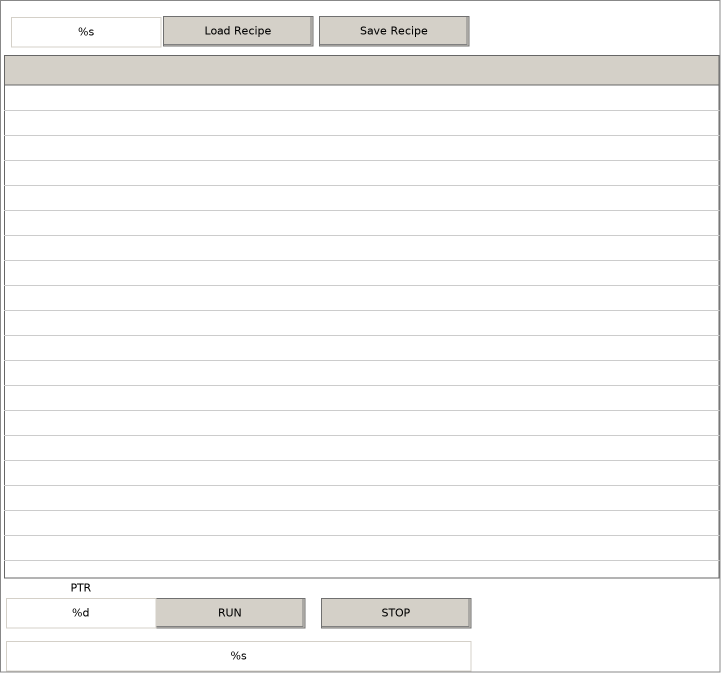
VISUALIZATION TempJozsiProg  // 721x673
    Button (163,16 150x30), "Load Recipe"
        OnMouseUp: execute {
            GVL.RecipeManagerCommands.LoadFromAndWriteRecipe('ProgramsJozsi','Ertekek',JozsiProcess.sRecipeName);
            JozsiProcess.bRunning:=FALSE;
            JozsiProcess.iPtr:=0;
        }
    Table (4,55 715x523), data array: JozsiProcess.asActualProgram
        p3854506369: JozsiProcess.asActualProgram[0,INDEX]
        p1892666644: JozsiProcess.asActualProgram[1,INDEX]
        p338671338: JozsiProcess.asActualProgram[2,INDEX]
        p2170511999: JozsiProcess.asActualProgram[3,INDEX]
        p3723444502: JozsiProcess.asActualProgram[4,INDEX]
        p1218418051: JozsiProcess.asActualProgram[5,INDEX]
        p2232123230: Parancs
        p511219082: Param1
        p1755163831: Param2
        p4092479075: Param3
        p2237128397: Param4
        p505689113: Param5
        Columns.Column.[2].Template: OnMouseClick: write the text variable via Edit
        Columns.Column.[0].Template: OnMouseClick: write the text variable via Edit
        Columns.Column.[1].Template: OnMouseClick: write the text variable via Edit
        Columns.Column.[4].Template: OnMouseClick: write the text variable via Edit
        Columns.Column.[3].Template: OnMouseClick: write the text variable via Edit
        Columns.Column.[5].Template: OnMouseClick: write the text variable via Edit
    Textfield (11,17 150x30), "%s", text variable: JozsiProcess.sRecipeName
        OnMouseClick: write the text variable via Edit
    Button (319,16 150x30), "Save Recipe"
        OnMouseUp: execute { GVL.RecipeManagerCommands.ReadAndSaveRecipeAs('ProgramsJozsi','Ertekek',JozsiProcess.sRecipeName); }
    Button (155,598 150x30), "RUN"
        OnMouseUp: execute { JozsiProcess.bRunning:=TRUE; }
    Button (321,598 150x30), "STOP"
        OnMouseUp: execute { JozsiProcess.bRunning:=FALSE; }
    Textfield (6,598 150x30), "%d", text variable: JozsiProcess.iPtr
        OnMouseClick: write the text variable via VisuDialogs.Numpad
    Label (6,573 150x30), "PTR"
    Textfield (6,641 465x30), "%s", text variable: JozsiProcess.asActualProgram[0,JozsiProcess.iPtr], input disabled if: TRUE
END_VISUALIZATION

(* stored: Version 1.1.0.1, ProductVersion 3.1.4024.11
   Visu TempJozsiProg: Id {8e0ada04-60b3-4fbd-a5ce-8ff586ae2efe} *)
